// TwinCAT 3 PLC project Projektbeispiel1
// ProgramVersion: 3.1.4023.0
// libraries:
//   Tc2_Math, * (Beckhoff Automation GmbH)
//   Tc2_Standard, * (Beckhoff Automation GmbH)
//   Tc2_System, * (Beckhoff Automation GmbH)
//   Tc3_Module, * (Beckhoff Automation GmbH)
//   Tc2_Utilities,3.3.38.0,Beckhoff Automation GmbH
//   Util,3.5.11.0,System
// project tree:
//   / PlcTask.TcTTO
//   POUs/ MAIN.TcPOU, POU.TcPOU
// real-time tasks:
//   TASK PlcTask: cycle T#10ms, priority 20, ADS port 350
// I/O:
//   DEVICE Gerät 2 (EtherCAT), AmsNetId 5.84.115.177.3.1
//     Klemme 1 (EK1200) [EK1200-5000 EtherCAT Netzteil (2A E-Bus)]
//       Klemme 2 (EL1008) [EL1008 8K. Dig. Eingang 24V, 3ms]
//       Klemme 3 (EL2008) [EL2008 8K. Dig. Ausgang 24V, 0.5A]
//       Klemme 4 (EL3208-0010) [EL3208-0010 8K. Ana. Eingang PT1000 (RTD)]
//       Klemme 5 (EL9011) [EL9011 Endklemme]
// variable links:
//   Projektbeispiel1/Projektbeispiel1 Instance <-> Device 2 (EtherCAT)/Term 1 (EK1200)/Term 2 (EL1008)
//     PlcTask Inputs/POU.i3 <-> Channel 3/Input
//   Projektbeispiel1/Projektbeispiel1 Instance <-> Device 2 (EtherCAT)/Term 1 (EK1200)/Term 3 (EL2008)
//     PlcTask Outputs/MAIN.Sfertig <-> Channel 2/Output
//     PlcTask Outputs/POU.a{3..8} <-> Channel {3..8}/Output  (6 links)
//   Projektbeispiel1/Projektbeispiel1 Instance <-> Device 2 (EtherCAT)/Term 1 (EK1200)/Term 4 (EL3208-0010)
//     PlcTask Inputs/MAIN.Temperatur <-> RTD Inputs Channel 1/Value

CONFIGURATION Projektbeispiel1
    RESOURCE PLC ON TwinCAT3
        TASK PlcTask(INTERVAL := T#10ms, PRIORITY := 20);
        PROGRAM MAIN WITH PlcTask : MAIN;
    END_RESOURCE
END_CONFIGURATION

// ---- POUs/MAIN.TcPOU
PROGRAM MAIN
VAR
	//bInput1 AT %I*: BOOL;
	//bOutput2 AT %Q*:BOOL;
	bBackhofengedruckt :BOOL;
	Sfertig AT %Q* :BOOL;
	fbtimer AT %I* :TP;
	fbtrigger :R_TRIG;
	Anzahlpizza:DINT;
	testBit:BOOL;
Temperatur AT %I*: INT;
angezeigterWert:LREAL;
angezeigterWert1:INT;
angezeigterWert2:REAL;
Temperatureanzeige:STRING;





	
	
END_VAR

//bOutput2:=NOT bInput1;
angezeigterWert:=INT_TO_REAL(Temperatur)/100;
//angezeigterWert1:=REAL_TO_INT(angezeigterWert*100);
//angezeigterWert2:=INT_TO_REAL(angezeigterWert1/100);
temperatureanzeige:=LREAL_TO_FMTSTR(angezeigterWert, 2, TRUE);
	
	
fbtimer(IN:=bBackhofengedruckt, PT:=T#5S);
	Sfertig:=fbtimer.Q;
fbtrigger(clk:=Sfertig);
IF fbtrigger.Q THEN
	Anzahlpizza:= Anzahlpizza+1;
	//angezeigterWert:=INT_TO_REAL(Temperatur)/100;
	//angezeigterWert:= temperatur/100;
	
END_IF

pou();

END_PROGRAM

// ---- POUs/POU.TcPOU
PROGRAM POU
VAR
	fbtimer1:TOF;
	rs:RS;
	BLINK1 :BLINK;
	TIMELOW:TIME;
	Initialschritt:SR;
	Schritt1:SR;
	Schritt2:SR;
	Schritt3:SR;
	Schritt4:SR;
	Schritt5:SR;

	
	
END_VAR

VAR_INPUT
	i3 AT %I*:BOOL;
	i4 AT %I*:BOOL;
	i5 AT %I*:BOOL;
	i6 AT %I*:BOOL;
	i7 AT %I*:BOOL;
END_VAR
VAR_OUTPUT
	a2 AT %Q*: BOOL;
	a3 AT %Q*: BOOL;
	a4 AT %Q*: BOOL;
	a5 AT %Q*: BOOL;
	a6 AT %Q*: BOOL;
	a7 AT %Q*: BOOL;
	a8 AT %Q*: BOOL;
END_VAR

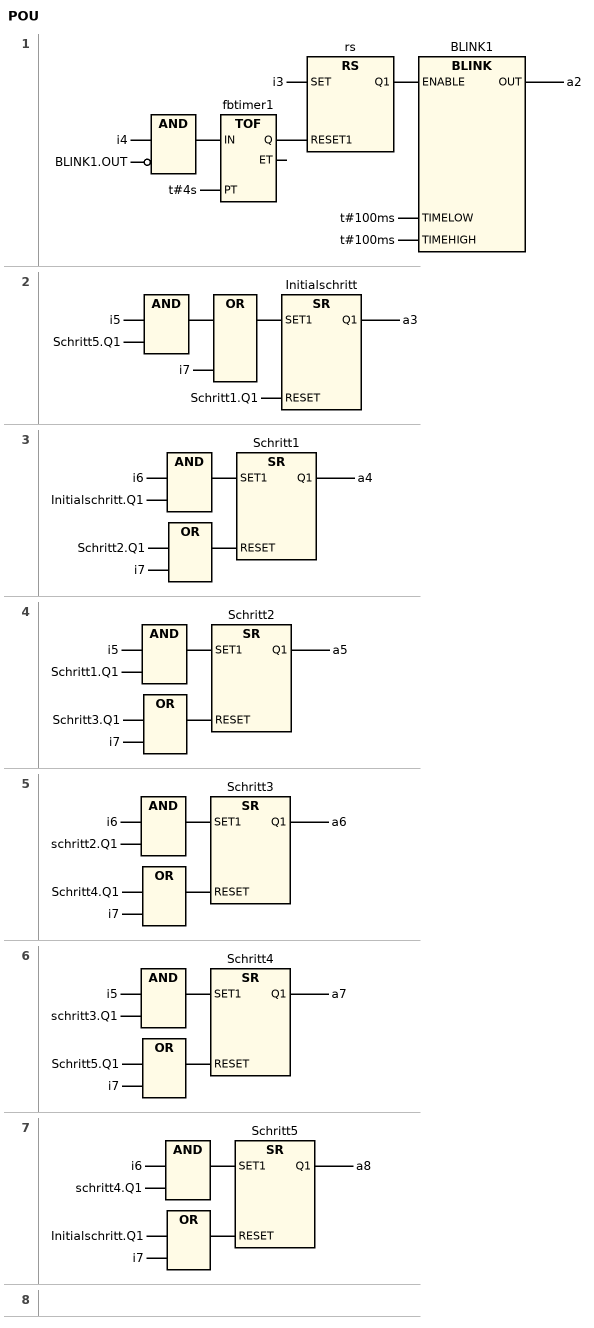
// NETWORK 1
fbtimer1(IN := i4 AND NOT BLINK1.OUT, PT := t#4s); // TOF
rs(SET := i3, RESET1 := fbtimer1.Q);
BLINK1(ENABLE := rs.Q1, TIMELOW := t#100ms, TIMEHIGH := t#100ms); // BLINK
a2 := BLINK1.OUT;

// NETWORK 2
Initialschritt(SET1 := i5 AND Schritt5.Q1 OR i7, RESET := Schritt1.Q1); // SR
a3 := Initialschritt.Q1;

// NETWORK 3
Schritt1(SET1 := i6 AND Initialschritt.Q1, RESET := Schritt2.Q1 OR i7); // SR
a4 := Schritt1.Q1;

// NETWORK 4
Schritt2(SET1 := i5 AND Schritt1.Q1, RESET := Schritt3.Q1 OR i7); // SR
a5 := Schritt2.Q1;

// NETWORK 5
Schritt3(SET1 := i6 AND schritt2.Q1, RESET := Schritt4.Q1 OR i7); // SR
a6 := Schritt3.Q1;

// NETWORK 6
Schritt4(SET1 := i5 AND schritt3.Q1, RESET := Schritt5.Q1 OR i7); // SR
a7 := Schritt4.Q1;

// NETWORK 7
Schritt5(SET1 := i6 AND schritt4.Q1, RESET := Initialschritt.Q1 OR i7); // SR
a8 := Schritt5.Q1;

// NETWORK 8

END_PROGRAM
